// TIA Portal V20 export
VAR_GLOBAL   // PLC tag table "VALVE_TAGS"
END_VAR
VAR_GLOBAL CONSTANT   // user constants
   "V-10101" : String := 'V-10101';   // Unit 1 Module 1 main inlet valve
   "V-10102" : String := 'V-10102';   // Unit 1 Module 1 secondary inlet valve
   "V-10103" : String := 'V-10103';   // Unit 1 Module 1 drain valve
   "V-10104" : String := 'V-10104';   // Unit 1 Module 1 bypass valve
   "V-10201" : String := 'V-10201';   // Unit 1 Module 2 tank outlet
   "V-10202" : String := 'V-10202';   // Unit 1 Module 2 product transfer
   "V-10111" : String := 'V-10111';   // Unit 1 module 1 valve 1 (instance 1)
   "V-10112" : String := 'V-10112';   // Unit 1 module 1 valve 1 (instance 2)
   "V-10113" : String := 'V-10113';   // Unit 1 module 1 valve 1 (instance 3)
   "V-10114" : String := 'V-10114';   // Unit 1 module 1 valve 1 (instance 4)
   "V-10121" : String := 'V-10121';   // Unit 1 module 1 valve 2 (instance 1)
   "V-10122" : String := 'V-10122';   // Unit 1 module 1 valve 2 (instance 2)
   "V-10123" : String := 'V-10123';   // Unit 1 module 1 valve 2 (instance 3)
   "V-10124" : String := 'V-10124';   // Unit 1 module 1 valve 2 (instance 4)
   "V-10131" : String := 'V-10131';   // Unit 1 module 1 valve 3 (instance 1)
   "V-10132" : String := 'V-10132';   // Unit 1 module 1 valve 3 (instance 2)
   "V-10133" : String := 'V-10133';   // Unit 1 module 1 valve 3 (instance 3)
   "V-10134" : String := 'V-10134';   // Unit 1 module 1 valve 3 (instance 4)
   "V-10211" : String := 'V-10211';   // Unit 1 module 2 valve 1 (instance 1)
   "V-10212" : String := 'V-10212';   // Unit 1 module 2 valve 1 (instance 2)
   "V-10213" : String := 'V-10213';   // Unit 1 module 2 valve 1 (instance 3)
   "V-10214" : String := 'V-10214';   // Unit 1 module 2 valve 1 (instance 4)
   "V-10221" : String := 'V-10221';   // Unit 1 module 2 valve 2 (instance 1)
   "V-10222" : String := 'V-10222';   // Unit 1 module 2 valve 2 (instance 2)
   "V-10223" : String := 'V-10223';   // Unit 1 module 2 valve 2 (instance 3)
   "V-10224" : String := 'V-10224';   // Unit 1 module 2 valve 2 (instance 4)
   "V-10231" : String := 'V-10231';   // Unit 1 module 2 valve 3 (instance 1)
   "V-10232" : String := 'V-10232';   // Unit 1 module 2 valve 3 (instance 2)
   "V-10233" : String := 'V-10233';   // Unit 1 module 2 valve 3 (instance 3)
   "V-10234" : String := 'V-10234';   // Unit 1 module 2 valve 3 (instance 4)
   "V-20111" : String := 'V-20111';   // Unit 2 module 1 valve 1 (instance 1)
   "V-20112" : String := 'V-20112';   // Unit 2 module 1 valve 1 (instance 2)
   "V-20113" : String := 'V-20113';   // Unit 2 module 1 valve 1 (instance 3)
   "V-20114" : String := 'V-20114';   // Unit 2 module 1 valve 1 (instance 4)
   "V-20121" : String := 'V-20121';   // Unit 2 module 1 valve 2 (instance 1)
   "V-20122" : String := 'V-20122';   // Unit 2 module 1 valve 2 (instance 2)
   "V-20123" : String := 'V-20123';   // Unit 2 module 1 valve 2 (instance 3)
   "V-20124" : String := 'V-20124';   // Unit 2 module 1 valve 2 (instance 4)
   "V-20131" : String := 'V-20131';   // Unit 2 module 1 valve 3 (instance 1)
   "V-20132" : String := 'V-20132';   // Unit 2 module 1 valve 3 (instance 2)
   "V-20133" : String := 'V-20133';   // Unit 2 module 1 valve 3 (instance 3)
   "V-20134" : String := 'V-20134';   // Unit 2 module 1 valve 3 (instance 4)
   "V-20211" : String := 'V-20211';   // Unit 2 module 2 valve 1 (instance 1)
   "V-20212" : String := 'V-20212';   // Unit 2 module 2 valve 1 (instance 2)
   "V-20213" : String := 'V-20213';   // Unit 2 module 2 valve 1 (instance 3)
   "V-20214" : String := 'V-20214';   // Unit 2 module 2 valve 1 (instance 4)
   "V-20221" : String := 'V-20221';   // Unit 2 module 2 valve 2 (instance 1)
   "V-20222" : String := 'V-20222';   // Unit 2 module 2 valve 2 (instance 2)
   "V-20223" : String := 'V-20223';   // Unit 2 module 2 valve 2 (instance 3)
   "V-20224" : String := 'V-20224';   // Unit 2 module 2 valve 2 (instance 4)
   "V-20231" : String := 'V-20231';   // Unit 2 module 2 valve 3 (instance 1)
   "V-20232" : String := 'V-20232';   // Unit 2 module 2 valve 3 (instance 2)
   "V-20233" : String := 'V-20233';   // Unit 2 module 2 valve 3 (instance 3)
   "V-20234" : String := 'V-20234';   // Unit 2 module 2 valve 3 (instance 4)
END_VAR
